TYPE ST_AxisHaltParameter EXTENDS ST_AxisStopParameter :
STRUCT
	eBufferMode: MC_BufferMode := MC_Aborting;
END_STRUCT
END_TYPE

(* stored: Version 1.1.0.1, ProductVersion 3.1.4022.9
   DUT ST_AxisHaltParameter: Id {eab622aa-f8ed-4282-9086-c443211dcdc3} *)
